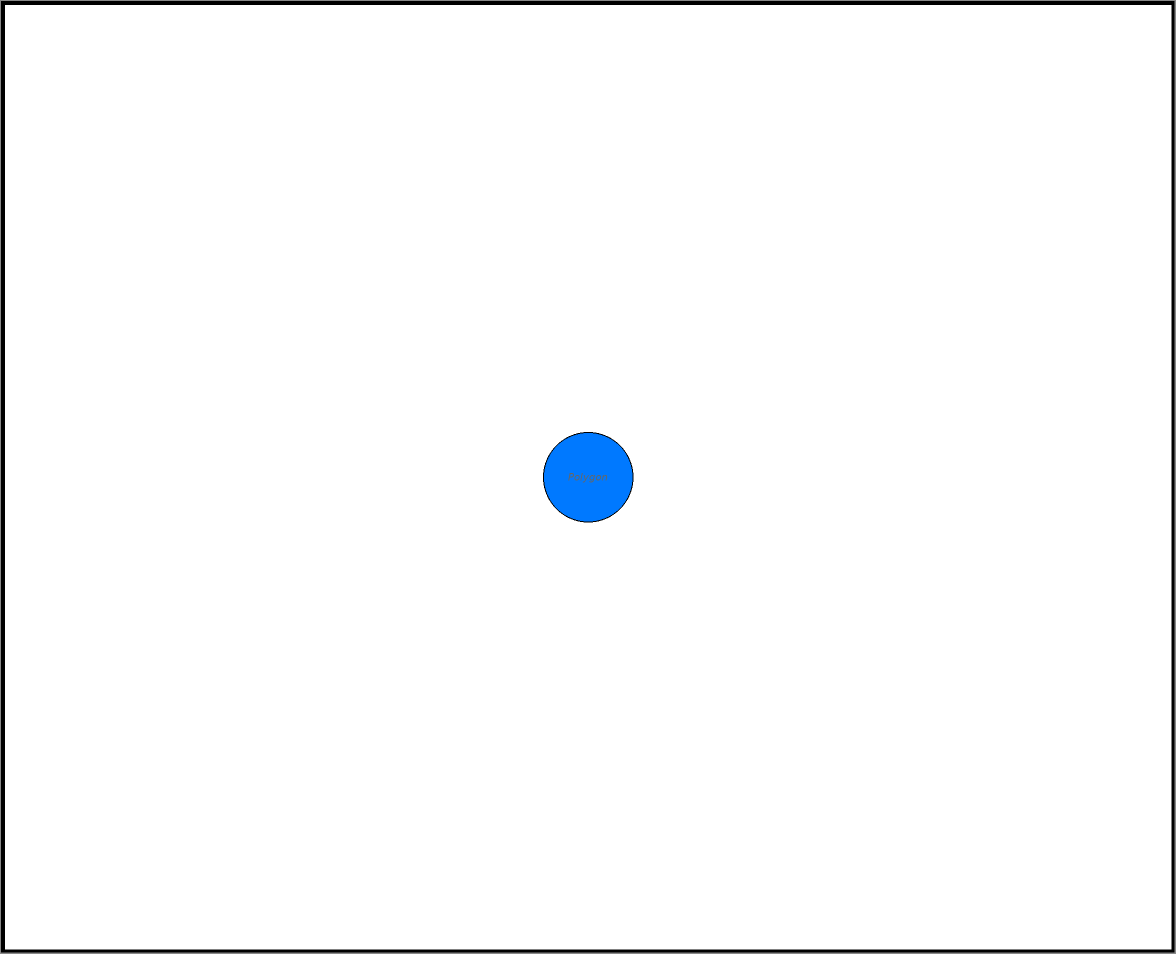
VISUALIZATION FigurePlayerDisplay  // 1176x954
    Rectangle (0,0 1176x954)
    Ellipse (543,432 90x90), invisible if: NOT Touchpanel.bContactAvailable
        p3560616238: Touchpanel.touch_scale_x.rX_mm*3
        p2738717112: -Touchpanel.touch_scale_y.rX_mm*3
    Frame (0,0 1176x954)
        shows Polygon(pVisu := CONTROLLER.FB_FigurePlayer_0.pFigure^.pVisu, VisuLenght := CONTROLLER.FB_FigurePlayer_0.pFigure^.VisuLenght)
END_VISUALIZATION

(* stored: Version 1.1.0.1, ProductVersion 3.1.4024.12
   Visu FigurePlayerDisplay: Id {e7069c83-2044-49b7-a6c7-86a4bbc06f25} *)
